PROGRAM MAIN
VAR
	fbModbusTCP: FB_Modbus_TCP_Client;
END_VAR

fbModbusTCP(
	sIPAddress:= , 
	uiTCPPort:=502 , 
	byUnitID:=255 , 
	iFunctionNo:= , 
	wAddress:= , 
	stData:= , 
	uiQuantity:= , 
	bExecute:= , 
	tTimeout:= , 
	bReset:= , 
	nValue:= , 
	bBusy=> , 
	bError=> , 
	udiErrorId=> , 
	bDone=> );

END_PROGRAM

(* stored: Version 1.1.0.1, ProductVersion 3.1.4024.15
   POU MAIN: Id {6066e2c5-f7ce-4fbe-9c73-fceb74d3e585}, SpecialFunc None *)
